FUNCTION_BLOCK FB_SATTTest EXTENDS FB_TestSuite
VAR

    axRef    : AXIS_REF;
    fbPDS    : LCLS_Tc_DevAbs.FB_PersistentDataStorage;

    fbMotorY      : FB_MotionStageNC(AxisRef := axRef, iPersistentDataStorage := fbPDS, sName := 'Y');
    aiMotionStage : ARRAY[1..MotionConstants.MAX_STATE_MOTORS] OF I_MotionStage := [fbMotorY];

    {attribute 'pytmc' := '
        pv: MMS
        array: 1..1 | 1..9
    '}
    astPositionState : ARRAY[1..MotionConstants.MAX_STATE_MOTORS]
                         OF ARRAY[1..GeneralConstants.MAX_STATES] OF ST_PositionState;

    fbFFHWO : FB_HardwareFFOutput;

    sDeviceName : STRING := 'AT1K4:L2SI';
    bFileReaderBusy :  BOOL;
    fbArbiter  : FB_Arbiter(1);
    fbSubSysIO : FB_DummyArbIO;

    fbSATT : FB_SXR_SATT_Stage(
        aiMotionStage    := aiMotionStage,
        astPositionState := astPositionState,
        fbFFHWO          := fbFFHWO,
        bFileReaderBusy  := bFileReaderBusy,
        sDeviceName      := sDeviceName,
        RTDPMPSState     := 'AT1K4:L2SI-RTD'
    );

    stDefault : ST_PositionState := (
        fDelta        := 0.2,
        bMoveOk       := TRUE,
        bValid        := TRUE,
        bUseRawCounts := FALSE
    );

    afbStateDefaults : ARRAY[1..9] OF FB_CC_StateDefaultsConfig[
        (stPositionState := astPositionState[1][E_SXR_SATT_Position.OUT],     stDefault := stDefault, sName := 'Out',     fPosition := 10),
        (stPositionState := astPositionState[1][E_SXR_SATT_Position.FILTER1], stDefault := stDefault, sName := 'Filter1', fPosition := 20),
        (stPositionState := astPositionState[1][E_SXR_SATT_Position.FILTER2], stDefault := stDefault, sName := 'Filter2', fPosition := 30),
        (stPositionState := astPositionState[1][E_SXR_SATT_Position.FILTER3], stDefault := stDefault, sName := 'Filter3', fPosition := 40),
        (stPositionState := astPositionState[1][E_SXR_SATT_Position.FILTER4], stDefault := stDefault, sName := 'Filter4', fPosition := 50),
        (stPositionState := astPositionState[1][E_SXR_SATT_Position.FILTER5], stDefault := stDefault, sName := 'Filter5', fPosition := 60),
        (stPositionState := astPositionState[1][E_SXR_SATT_Position.FILTER6], stDefault := stDefault, sName := 'Filter6', fPosition := 70),
        (stPositionState := astPositionState[1][E_SXR_SATT_Position.FILTER7], stDefault := stDefault, sName := 'Filter7', fPosition := 80),
        (stPositionState := astPositionState[1][E_SXR_SATT_Position.FILTER8], stDefault := stDefault, sName := 'Filter8', fPosition := 90)
    ];

    (* Per-filter material + thickness (integrator-owned) written into
       the device's arrFilters table via FB_SATT_FilterConfig. *)
    afbFilterCfg : ARRAY[1..8] OF FB_SATT_FilterConfig[
        (stFilter := fbSATT.arrFilters[1], sFilterMaterial := 'C',  fFilterThickness_um := 25),
        (stFilter := fbSATT.arrFilters[2], sFilterMaterial := 'C',  fFilterThickness_um := 50),
        (stFilter := fbSATT.arrFilters[3], sFilterMaterial := 'C',  fFilterThickness_um := 100),
        (stFilter := fbSATT.arrFilters[4], sFilterMaterial := 'Si', fFilterThickness_um := 200),
        (stFilter := fbSATT.arrFilters[5], sFilterMaterial := 'Si', fFilterThickness_um := 320),
        (stFilter := fbSATT.arrFilters[6], sFilterMaterial := 'Si', fFilterThickness_um := 640),
        (stFilter := fbSATT.arrFilters[7], sFilterMaterial := 'Si', fFilterThickness_um := 1280),
        (stFilter := fbSATT.arrFilters[8], sFilterMaterial := 'Si', fFilterThickness_um := 2560)
    ];

    bFirstScan : BOOL := TRUE;
    i          : UINT;
END_VAR

IF bFirstScan THEN
    fbMotorY.SetModeEnableLimits(
        LimBackward    := TRUE,
        LimForward     := TRUE,
        HomeEnable     := FALSE,
        BrakeMode      := E_StageBrakeMode.NO_BRAKE,
        EnableMode     := E_StageEnableMode.DURING_MOTION,
        HomeMode       := E_EpicsHomeCmd.NONE,
        UserEnable     := TRUE,
        HardwareEnable := TRUE
    );
    fbMotorY.SetVelocity(Velocity := 15.5);
    fbMotorY.RestoreMotionParams      := FALSE;
    fbMotorY.DoNotRestoreNcParameters := TRUE;
    bFirstScan := FALSE;
END_IF
// avoid a division by Zero in F_CalculateAbsorbptionConstant from Physics Library
// protection must be added there on neV
PMPS_GVL.stCurrentBeamParameters.neV := 250.0;
fbPDS();
fbMotorY();
fbSATT();
fbSubSysIO(LA := fbArbiter, FFO := fbFFHWO);

TestConfig();
TestStateMove();
TestTempFFO();

METHOD AssertBothTempFault
VAR_INPUT
    Message : STRING;
END_VAR

AssertFalse(
    fbSATT.fbRTD_1.FFO.i_xOK,
    CONCAT('SATT RTD1 expected fault: ', Message)
);
AssertFalse(
    fbSATT.fbRTD_2.FFO.i_xOK,
    CONCAT('SATT RTD2 expected fault: ', Message)
);
END_METHOD

METHOD AssertNeitherTempFault
VAR_INPUT
    Message : STRING;
END_VAR

AssertTrue(
    fbSATT.fbRTD_1.FFO.i_xOK,
    CONCAT('SATT RTD1 expected ok: ', Message)
);
AssertTrue(
    fbSATT.fbRTD_2.FFO.i_xOK,
    CONCAT('SATT RTD2 expected ok: ', Message)
);
END_METHOD

METHOD SetSATTTemp
VAR_INPUT
    iTempC : INT;
END_VAR
VAR
    ptr : POINTER TO INT;
END_VAR

ptr  := ADR(fbSATT.fbRTD_1.iRaw);
ptr^ := iTempC * 100;

ptr  := ADR(fbSATT.fbRTD_2.iRaw);
ptr^ := iTempC * 100;
END_METHOD

(*
    Verifies the integrator-side configurators each write their own
    slot fields exactly once at init, with no overlap:
      - FB_CC_StateDefaultsConfig -> sName, fPosition, and fDelta from
        the stDefault baseline
      - FB_SATT_FilterConfig      -> arrFilters material, thickness
    All are one-shot CallAfterInit writes, so the values are present
    from the first scan; this test asserts once and finishes.
*)
METHOD TestConfig
VAR CONSTANT
    fTol : LREAL := 0.001;
END_VAR
TEST('TestSATTConfig');

(* FB_CC_StateDefaultsConfig wrote sName + the fDelta baseline. *)
AssertTrue(
    astPositionState[1][E_SXR_SATT_Position.OUT].sName = 'Out',
    'OUT sName not set by FB_CC_StateDefaultsConfig');
AssertTrue(
    ABS(astPositionState[1][E_SXR_SATT_Position.OUT].fDelta - 0.2) <= fTol,
    'OUT fDelta not copied from stDefault by FB_CC_StateDefaultsConfig');
AssertTrue(
    astPositionState[1][E_SXR_SATT_Position.FILTER1].sName = 'Filter1',
    'FILTER1 sName not set by FB_CC_StateDefaultsConfig');

(* FB_CC_StateDefaultsConfig wrote fPosition. *)
AssertTrue(
    ABS(astPositionState[1][E_SXR_SATT_Position.OUT].fPosition - 10.0) <= fTol,
    'OUT fPosition not set by FB_CC_StateDefaultsConfig');
AssertTrue(
    ABS(astPositionState[1][E_SXR_SATT_Position.FILTER1].fPosition - 20.0) <= fTol,
    'FILTER1 fPosition not set by FB_CC_StateDefaultsConfig');

(* FB_SATT_FilterConfig wrote material + thickness into arrFilters. *)
AssertTrue(
    fbSATT.arrFilters[1].sFilterMaterial = 'C',
    'arrFilters[1] material not set by FB_SATT_FilterConfig');
AssertTrue(
    ABS(fbSATT.arrFilters[1].fFilterThickness_um - 25.0) <= fTol,
    'arrFilters[1] thickness not set by FB_SATT_FilterConfig');

TEST_FINISHED();
END_METHOD

(*
    Smoke test for SATT state-move wiring. Walks OUT then FILTER1 and
    asserts each lands within fTolerance of the configured fPosition.
    Mirrors FB_REFTest: stageReady gate up front, NOT bMoving +
    position-tolerance check per state, 60s watchdog, on timeout
    AssertTrue(FALSE, ...) with the current step and observed
    position. Two moves is enough to exercise the FB wiring; the
    motion stack itself is covered by the
    lcls-twincat-motion-abstraction test suite.
*)
METHOD TestStateMove
VAR_INST
    tonTimer  : TON;
    nTestStep : INT := 0;
    fObserved : LREAL;
END_VAR
VAR CONSTANT
    fTolerance : LREAL := 2.0;
END_VAR
TEST('TestSATTStateMove');

tonTimer(IN := TRUE, PT := T#60s);
fObserved := fbMotorY.stMotionStatus.fActPosition;

CASE nTestStep OF
    0:

        IF fbMotorY.stMotionStatus.bStageReady
           AND NOT fbMotorY.stMotionStatus.bError THEN
            fbSATT.eEnumSet := E_SXR_SATT_Position.OUT;
            nTestStep       := 1;
        END_IF
    1:
        (* OUT is configured at fPosition := 10 in afbStateDefaults[1]. *)
        IF fbSATT.eEnumGet = E_SXR_SATT_Position.OUT
           AND NOT fbMotorY.stMotionStatus.bMoving
           AND ABS(fObserved - 10.0) <= fTolerance THEN
            fbSATT.eEnumSet := E_SXR_SATT_Position.FILTER1;
            nTestStep       := 2;
        END_IF
    2:
        (* FILTER1 is configured at fPosition := 20 in afbStateDefaults[2]. *)
        IF fbSATT.eEnumGet = E_SXR_SATT_Position.FILTER1
           AND NOT fbMotorY.stMotionStatus.bMoving
           AND ABS(fObserved - 20.0) <= fTolerance THEN
            AssertTrue(
                Condition := TRUE,
                Message   := 'TestSATTStateMove: OUT then FILTER1 reached within tolerance');
            nTestStep := 3;
        END_IF
END_CASE

IF nTestStep = 3 THEN
    TEST_FINISHED();
ELSIF tonTimer.Q THEN
    AssertTrue(
        Condition := FALSE,
        Message   := CONCAT(
            CONCAT(
                CONCAT('TestSATTStateMove: timed out at step ', TO_STRING(nTestStep)),
                CONCAT(', eEnumGet=', TO_STRING(TO_UDINT(fbSATT.eEnumGet)))),
            CONCAT(', fActPos=', TO_STRING(fObserved))));
    TEST_FINISHED();
END_IF
END_METHOD

METHOD TestTempFFO
VAR_INST
    tonTimer    : TON;
    nStep       : UINT := 0;
    bOutChecked : BOOL := FALSE;
    bInChecked  : BOOL := FALSE;
END_VAR
VAR CONSTANT
    nLastStep : UINT := 3;
END_VAR

(* Do we fault at the correct times?
   Parasitically depends on state move test. *)
TEST('TestSATTTempFFO');

(* Prepare a timeout *)
tonTimer(IN := TRUE, PT := T#10s);

CASE nStep OF
    0:
        (* Set the thermocouple temperatures to crazy high number. *)
        SetSATTTemp(100);
        nStep := nStep + 1;
    1:
        (* Wait till we see "OUT" state and one other state (OUT
           should be no fault). *)
        IF fbSATT.eEnumGet = E_SXR_SATT_Position.OUT THEN
            AssertNeitherTempFault('was in out position');
            bOutChecked := TRUE;
        ELSIF fbSATT.eEnumGet <> E_SXR_SATT_Position.UNKNOWN THEN
            AssertBothTempFault('was in a target position');
            bInChecked := TRUE;
        END_IF
        IF bOutChecked AND bInChecked THEN
            nStep := nStep + 1;
        END_IF
    2:
        (* Set the thermocouple temperatures to low again. *)
        SetSATTTemp(0);
        nStep := nStep + 1;
    3:
        AssertNeitherTempFault('has low temp reading');
        nStep := nStep + 1;
END_CASE

IF tonTimer.Q OR nStep > nLastStep THEN
    AssertFalse(tonTimer.Q, 'Timeout in SATT temp FFO test');
    TEST_FINISHED();
END_IF
END_METHOD

END_FUNCTION_BLOCK

(* stored: Version 1.1.0.1
   POU FB_SATTTest: Id {383787d3-728f-42f6-950b-c99d26391aa0}, SpecialFunc None
   Method AssertBothTempFault: Id {95d6c1aa-c314-417f-8510-e65298bca360}
   Method AssertNeitherTempFault: Id {5de84732-353a-4a55-9eb9-df3ae8bca03b}
   Method SetSATTTemp: Id {7ebc7bb7-f0d1-456e-9851-f9318ff9a3aa}
   Method TestConfig: Id {c4e7a118-9f2b-4d63-8a07-3b5e6c1d2f44}
   Method TestStateMove: Id {6c59097f-e216-48c9-8846-19da78be43c4}
   Method TestTempFFO: Id {f4f8a550-63b6-47ea-b8a6-24727446e218} *)
